Staubli VAL3: userPage.pjx

--- userPage.pjx ---
Parameters version=s7.5 stackSize=5000 millimeterUnit=true
Program file=changeTrsf.pgx
Program file=changeValue.pgx
Program file=clear.pgx
Program file=divideString.pgx
Program file=editNumField.pgx
Program file=findPos.pgx
Program file=getListPosition.pgx
Program file=getMenu.pgx
Program file=getView.pgx
Program file=insertDialog.pgx
Program file=isListEmpty.pgx
Program file=leftPos.pgx
Program file=listadd.pgx
Program file=listcreate.pgx
Program file=listcursor.pgx
Program file=listdel.pgx
Program file=listempty.pgx
Program file=listevent.pgx
Program file=listframe.pgx
Program file=listins.pgx
Program file=listredraw.pgx
Program file=listupdate.pgx
Program file=midPos.pgx
Program file=nullKey.pgx
Program file=numCopy.pgx
Program file=printScroll.pgx
Program file=questionDialog.pgx
Program file=read.pgx
Program file=rightPos.pgx
Program file=scroll.pgx
Program file=selectNewField.pgx
Program file=setCenter.pgx
Program file=setMenu.pgx
Program file=setSizeList.pgx
Program file=setView.pgx
Program file=showBoolStatus.pgx
Program file=strfill.pgx
Program file=strfillchr.pgx
Program file=stringCopy.pgx
Program file=stringToArray.pgx
Program file=stringToFxArray.pgx
Program file=strlength.pgx
Program file=timerDialog.pgx
Program file=type.pgx
Program file=typeCenter.pgx
Program file=typeLen.pgx
Program file=typeMenu.pgx
Program file=yes_no.pgx
Program file=yes_no_cancel.pgx
Data file=userPage.dtx

--- userPage.dtx ---
bool Show
bool bReadWrite = true
public bool bShowDialog
public bool bUseEscape
public bool bUseRefresh
public num nBottomX[2]
  [0] = 17
  [1] = 17
public num nBottomY = 11
num nFirst
num nKey
num nOffSet
num nOldValue[2]
  [0] = 200
  [1] = 200
public num nPage = 10
public num nTopX[2]
  [0] = 21
  [1] = 21
public num nTopY
public num nView
public string sItems = "home"
string sMessage[3]
  [0] = "VALPLAST QUITTING..."
  [1] = " "
  [2] = "PLEASE WAIT"
public string sTitle = "HOME"

--- editNumField.pgx ---
public program editNumField(string x_sTitle, string& x_sItemName[], num& x_nItem[], num& x_nMin[], num& x_nMax[])
  local num j
  local num l_nSize
  local num l_nKey
  local string l_sEvent
  local num l_nIndex
  local num l_nField
  local string l_sItem
  local num i
  local string l_sEmpty
begin
  //
  // clear & copy
  //
  // nView=nFirst=0
  //call listempty()
  call numCopy(x_nItem,nOldValue)
  call numCopy(x_nItem,nOffSet)
  for j=0 to size(nOffSet)-1
    nOffSet[j]=0
  endFor
  // take the size
  l_nSize=size(x_nItem)-1
  // create the LIST
  call setSizeList(2,max((6-l_nSize/2)-2,2),34,min((l_nSize+1),8))
  call listcreate(x_sTitle)
  //
  // insert items
  //
  for j=0 to l_nSize
    l_sItem=x_sItemName[j]
    if l_sItem!=""
      call strlength(l_sItem,26)
      l_sItem=l_sItem+": "+toString(".1",x_nItem[j])
      call listadd(l_sItem)
      nOffSet[j]=nOffSet[max(j-1,0)]
    else
      nOffSet[j]=nOffSet[max(j-1,0)]+1
    endIf
  endFor
  // update the list
  call listupdate(0)
  do
    call clear(0,13)
    call typeMenu(8,"OK")
    l_nKey=get()
    call listevent(l_nKey,l_nIndex,l_sEvent)
    // use the offset
    i=l_nIndex+nOffSet[max(l_nIndex,0)]
    // on Enter Key
    if l_nKey==270
      call listcursor(l_nIndex,false)
      if size(x_nMin)==size(x_nItem)
        // use min and max
        l_sEmpty=""
        call changeValue(x_nItem[i],x_nMin[i],x_nMax[i],31,nView+nTopY+1,l_sEmpty)
      else
        call changeValue(x_nItem[i],x_nMin,x_nMax,31,nView+nTopY+1,l_sEmpty)
      endIf
      // UPDATE
      call listdel(l_nIndex)
      l_sItem=x_sItemName[i]
      call strlength(l_sItem,26)
      l_sItem=l_sItem+": "+toString(".1",x_nItem[i])
      call listins(l_sItem,l_nIndex)
      call listupdate(l_nIndex-nView)
    endIf
  until l_nKey==278 or l_nKey==255
  // escape use ?
  if l_nKey==255
    bUseEscape=true
    call numCopy(nOldValue,x_nItem)
  else
    bUseEscape=false
  endIf
  // exit
  call nullKey(l_nKey)
end

--- insertDialog.pgx ---
public program insertDialog(string x_sMsg, num& x_nItem[], num x_nMin, num x_nMax)
  local num l_nStartLine
  local num l_nLine
  local num i
  local num l_nPX
  local num l_nPY
  local string l_sItem
  local string l_sMessage
  local string l_sEmpty
begin
  //
  // modify the x_sItem, using a min max range
  //
  if watch(bShowDialog==false,3)==false
    bShowDialog=false
    return
  else
    setMutex(bShowDialog)
    // clear the line
    call clear(0,13)
    // look for the comma
    if round(x_nItem)!=x_nItem
      l_sItem=toString(".2",x_nItem)
    else
      l_sItem=toString("",x_nItem)
    endIf
    // print the line
    l_sItem=x_sMsg+">"+l_sItem
    call stringCopy(l_sItem,sMessage)
    // divide the sentence
    call divideString(sMessage,l_nLine)
    l_nStartLine=round(5-l_nLine/2)
    // Start LINE
    call type(0,l_nStartLine-2,"┌──────────────────────────────────────┐")
    call type(0,l_nStartLine-1,"│                                      │")
    // write the message
    for i=0 to l_nLine
      //call type(,"                                      ")
      l_sMessage=sMessage[i]
      call typeCenter(i+l_nStartLine,l_sMessage,38,false)
      call type(0,l_nStartLine+i,"│"+l_sMessage+"│")
    endFor
    // end LINE
    call type(0,l_nStartLine+l_nLine+1,"│                                      │")
    call type(0,l_nStartLine+l_nLine+2,"└──────────────────────────────────────┘")
    l_nPX=find(l_sMessage,">")+2
    l_nPY=l_nStartLine+l_nLine
    // change the value
    call changeValue(x_nItem,x_nMin,x_nMax,l_nPX,l_nPY,l_sEmpty)
    //
    bShowDialog=false
    bUseRefresh=true
    //
  endIf
end

--- listcreate.pgx ---
public program listcreate(string x_sTitle)
begin
  //
  // Staubli Copyright 2003 07 31
  //
  sTitle=x_sTitle
  call listframe(sTitle,nTopX,nTopY,nBottomX,nBottomY)
  call listempty()
end

--- listevent.pgx ---
public program listevent(num pkey (dimensions=1), num& pIndex[] (dimensions=1), string& pItem[] (dimensions=1))
  local num lVal
  local num l_nSize
  local bool l_bEmpty
begin
  //
  // Toneage Staubli product
  //
  //
  // get the item in the list and scroll it
  //
  call isListEmpty(l_bEmpty)
  // not allowed negative value
  nView=max(0,nView)
  nFirst=max(0,nFirst)
  pIndex=max(0,pIndex)
  // look for the empty
  if !l_bEmpty
    l_nSize=size(sItems)-1
    // check the overFlow
    l_nSize=size(sItems)-1
    if (nFirst+nView>l_nSize)
      // reset the value
      nFirst=nView=0
    endIf
    // security...
    switch (pkey)
      //Up
      case 261
        if ((nView-1)>=0)
          // no need to scroll only change cursor position
          call listcursor(nView,false)
          nView=nView-1
          call listcursor(nView,true)
          // print the scroll
          //call printScroll()
        else
          if nView==0
            // scroll up
            if ((nFirst-1)>=0)
              nFirst=nFirst-1
              call listupdate(nFirst)
            else
              // go to the end
              if nView+nFirst!=l_nSize
                call listcursor(nView,false)
                call selectNewField(l_nSize,nFirst+nView,nView)
              endIf
            endIf
          endIf
        endIf
      break
      //Down
      case 266
        if ((nView+nFirst+1)<size(sItems))
          // no need to scroll only chenge cursor position
          if ((nView+1)<nBottomY)
            call listcursor(nView,false)
            nView=nView+1
            call listcursor(nView,true)
            // print the scroll
            //call printScroll()
          else
            // move UP
            nFirst=nFirst+1
            call listupdate(nFirst)
          endIf
        else
          // go to the top
          if !(nView==0 and nFirst==0)
            call listcursor(nView,false)
            nView=0
            call listupdate(0)
          endIf
        endIf
      break
      //Page Up
      case 262
        if !(nView==0 and nFirst==0)
          call listcursor(nView,false)
          if ((nFirst+nView-nBottomY)>=0)
            // move one page up
            call selectNewField(nFirst+nView-nBottomY,nFirst+nView,nView)
          else
            // go to home
            nView=0
            call listupdate(0)
          endIf
        endIf
      break
      //Page Down
      case 267
        if nView+nFirst!=l_nSize
          call listcursor(nView,false)
          if ((nView+nFirst+nBottomY)<size(sItems)-1)
            // move one page down
            call selectNewField(nFirst+nView+nBottomY,nFirst+nView,nView)
          else
            // go to the end
            call selectNewField(l_nSize,nFirst+nView,nView)
          endIf
        endIf
      break
      //End
      case 269
        if nView+nFirst!=l_nSize
          // move to end
          call listcursor(nView,false)
          call selectNewField(l_nSize,nFirst+nView,nView)
        endIf
      break
      //Home
      case 265
        if !(nView==0 and nFirst==0)
          // move to home
          call listcursor(nView,false)
          nView=0
          call listupdate(0)
        endIf
      break
      default
      break
    endSwitch
    pIndex=nFirst+nView
    pItem=sItems[pIndex]
    //
  else
    // reset the item
    pItem=""
    pIndex=0
  endIf
end

--- listupdate.pgx ---
public program listupdate(num pFirst)
  local num lI
  local num lLen
  local string lStr
  local string lStr2
  local num lValue
  local num lView
  local num lX
  local num lY
  local num l_nSize
  local bool l_bEmpty
begin
  //
  // insert into the box all the data
  //
  // to prevent a negative value
  if pFirst>0
    nFirst=pFirst
  else
    nFirst=0
  endIf
  // save the coordinate
  lValue=nBottomY-1
  // check the overFlow
  l_nSize=size(sItems)-1
  if (nFirst+nView>l_nSize)
    // reset the value
    nFirst=nView=0
  endIf
  lI=0
  // check the unKnow poblem
  if l_nSize<lValue
    if nFirst!=0
      nView=nView+nFirst
      nFirst=0
    endIf
  endIf
  do
    lX=nTopX+1
    lY=nBottomY+lI-1
    lY=nTopY+lI+1
    lLen=nBottomX
    if ((lI+nFirst)<size(sItems))
      // print the item
      if (l_nSize>=0)
        lStr=mid(sItems[(lI+nFirst)],lLen,0)
      endIf
    else
      // print the blank line
      lStr="                                        "
    endIf
    // fill the line
    call strfill(lStr,lLen,lStr2)
    gotoxy(lX,lY)
    put(lStr2)
    lI=lI+1
  until (lI>lValue)
  // underlien the actual line
  call isListEmpty(l_bEmpty)
  if !l_bEmpty
    call listcursor(nView,true)
  else
    call listcursor(nView,false)
    nView=0
    nFirst=0
  endIf
  // print the scroll
  call printScroll()
end

--- nullKey.pgx ---
public program nullKey(num& x_nKey[])
begin
  wait(getKey()==-1)
  x_nKey=0
end

--- questionDialog.pgx ---
public program questionDialog(string x_sMsg, string& x_sButton[], num& x_nResult[])
  local bool lExit
  local num nLine
  local num i
  local num nStartLine
  local string l_sMessage
begin
  //---------------------------------
  //      D I A L O G    B O X
  //---------------------------------
  //
  // Show one dialog box. with an confirm question
  //
  if watch(bShowDialog==false,3)==false
    bShowDialog=false
    return
  else
    setMutex(bShowDialog)
    //
    //
    if x_sMsg!=""
      call stringCopy(x_sMsg,sMessage)
      call divideString(sMessage,nLine)
      nStartLine=round(5-nLine/2)
      // Start LINE
      call type(0,nStartLine-2,"┌──────────────────────────────────────┐")
      call type(0,nStartLine-1,"│                                      │")
      // write the message
      for i=0 to nLine
        l_sMessage=sMessage[i]
        call typeCenter(i+nStartLine,l_sMessage,38,false)
        call type(0,nStartLine+i,"│"+l_sMessage+"│")
      endFor
      // end LINE
      call type(0,nStartLine+nLine+1,"│                                      │")
      call type(0,nStartLine+nLine+2,"└──────────────────────────────────────┘")
    endIf
    // write the button message
    call clear(0,13)
    for i=0 to size(x_sButton)-1
      call typeMenu(8-i,x_sButton[i])
    endFor
    lExit=false
    x_nResult=-100
    do
      nKey=get()
      switch (nKey)
        case 270
          x_nResult=0
        break
        case 255
          x_nResult=-1
          bUseEscape=true
        break
        default
          // look if the button press is defined
          if (nKey>=271 and nKey<=278) and ((279-nKey)<=size(x_sButton))
            if x_sButton[278-nKey]!=""
              x_nResult=279-nKey
            endIf
          endIf
        break
      endSwitch
    until (x_nResult!=-100)
    //
    call nullKey(nKey)
    if x_nResult!=-1
      bUseEscape=false
    endIf
    //
    // release
    bShowDialog=false
    bUseRefresh=true
  endIf
end
